// TIA Portal V20 export
TYPE "LBP_typeMcp310AdditionalInput"
TITLE = MCP 310 image / Image du MCP 310
// Additional input image of MCP 310 / Image d'entrée supplémentaire du MCP 310
   STRUCT
      directKey1 : Bool;   // DT1
      directKey2 : Bool;   // DT2
      directKey3 : Bool;   // DT3
      directKey4 : Bool;   // DT4
      directKey5 : Bool;   // DT5
      directKey6 : Bool;   // DT6
      directKey7 : Bool;   // DT7
      directKey8 : Bool;   // DT8
      directKey9 : Bool;   // DT9
      directKey10 : Bool;   // DT10
      directKey11 : Bool;   // DT11
      directKey12 : Bool;   // DT12
      directKey13 : Bool;   // DT13
      directKey14 : Bool;   // DT14
      directKey15 : Bool;   // DT15
      directKey16 : Bool;   // DT16
      reserved2 : Byte;
      feedrateOvrA : Bool;
      feedrateOvrB : Bool;
      feedrateOvrC : Bool;
      feedrateOvrD : Bool;
      feedrateOvrE : Bool;
      reserved35 : Bool;
      reserved36 : Bool;
      reserved37 : Bool;
      spindleOvrA : Bool;
      spindleOvrB : Bool;
      spindleOvrC : Bool;
      spindleOvrD : Bool;
      spindleOvrE : Bool;
      reserved45 : Bool;
      reserved46 : Bool;
      reserved47 : Bool;
   END_STRUCT;
END_TYPE
